FUNCTION_BLOCK Valve (* Composite Function Block Type *)
  (* Standard: 61499-2 *)
  (* Version 0.0, 2011-12-21, 4DIAC-IDE, 4DIAC-Consortium *)
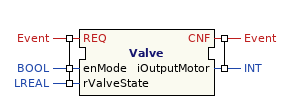
  EVENT_INPUT
    REQ WITH enMode, rValveState; (* Normal Execution Request *)
  END_EVENT
  EVENT_OUTPUT
    CNF WITH iOutputMotor; (* Execution Confirmation *)
  END_EVENT
  VAR_INPUT
    enMode : BOOL; (* Input event qualifier *)
    rValveState : LREAL;
  END_VAR
  VAR_OUTPUT
    iOutputMotor : INT; (* Output event qualifier *)
  END_VAR
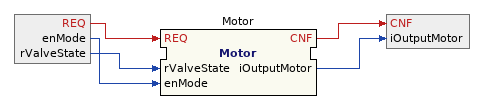
  FBS
    Motor : Motor;
  END_FBS
  EVENT_CONNECTIONS
    REQ TO Motor.REQ;
    Motor.CNF TO CNF;
  END_CONNECTIONS
  DATA_CONNECTIONS
    rValveState TO Motor.rValveState;
    enMode TO Motor.enMode;
    Motor.iOutputMotor TO iOutputMotor;
  END_CONNECTIONS
END_FUNCTION_BLOCK
